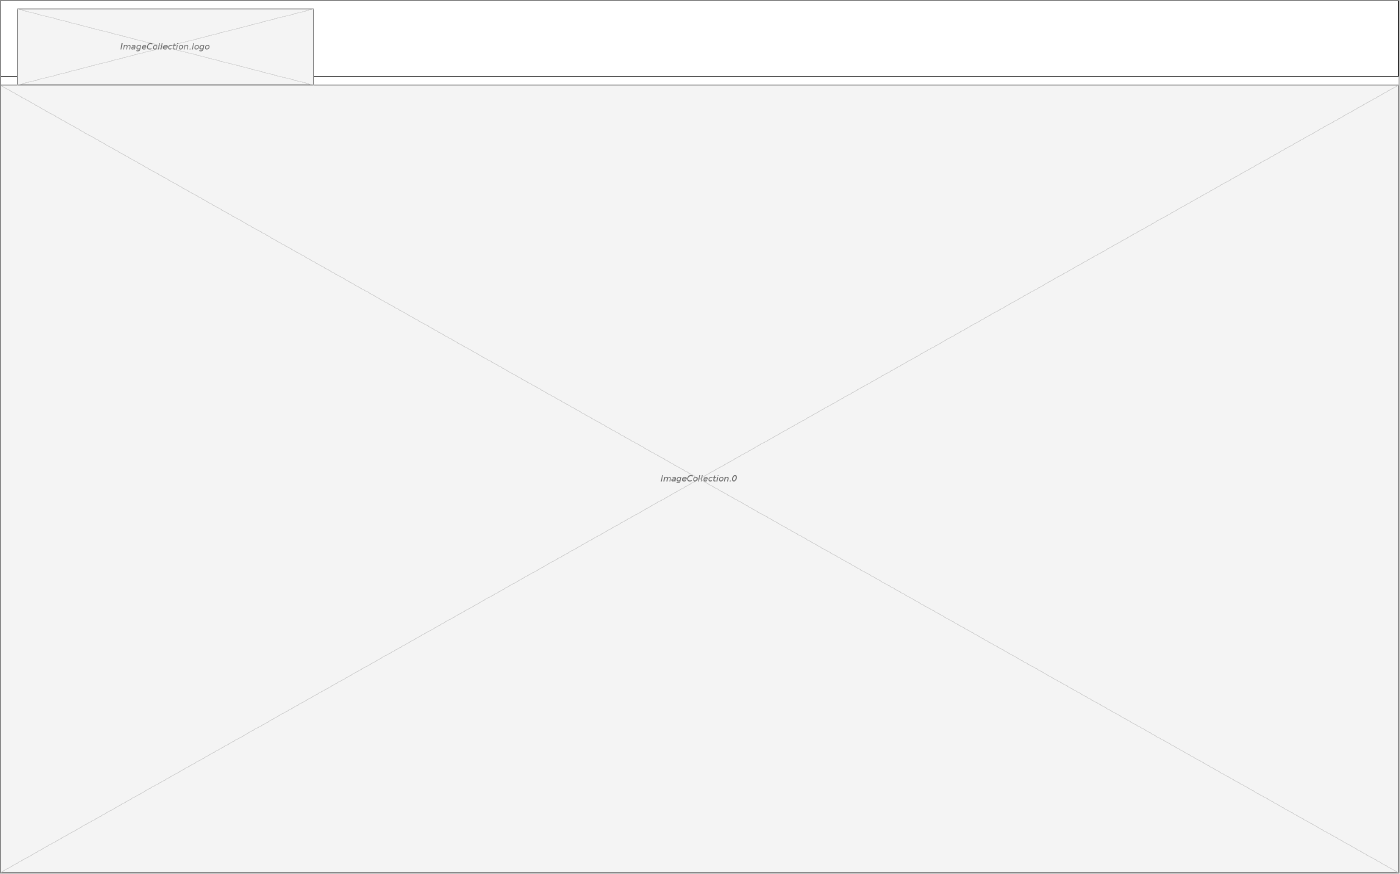
VISUALIZATION startView  // 1652x1032
    Rectangle (0,0 1650x90)
    Image (0,100 1650x930), image: ImageCollection.0
        OnMouseClick: change screen: AutomaticMode
        OnMouseClick: toggle bStartViewPressed
    Image (20,10 350x90), image: ImageCollection.logo
END_VISUALIZATION

(* stored: Version 1.1.0.1, ProductVersion 3.1.4018.2
   Visu startView: Id {8885aaf6-35ff-4925-b698-9167ed554e41} *)
